TYPE ST_WP_Stellwert :
STRUCT
	Betrieb		: BOOL;
	Freigabe	: BOOL;
	Modus		: SINT;
	WP_Stellung : BOOL;
END_STRUCT
END_TYPE

(* stored: Version 1.1.0.1, ProductVersion 3.1.4024.9
   DUT ST_WP_Stellwert: Id {81087e7f-3ccc-47d0-9e9f-114a3eaad616} *)
